(* CoDeSys 2.3 export: GLOBAL_CONSTANTS_PK.EXP *)

(* Global variable list: Global_Constants *)
VAR_GLOBAL CONSTANT

	gc_bHARTMaxModules		: BYTE := 16;		(* controller specific max. count of  mailbox io-modules *)

END_VAR
